# B&R Automation Studio project SimuladorTesis
Automation Studio 4.8.2.72; technology packages: mapp 5.8.0

## Configuration Config1

CPU X20CP1584, AutomationRuntime C4.90, Build 4.1.2, Safety 0.0, Vc V4.72.2

### Task classes (Cpu.sw)
```
Cyclic#2:
  MainLogic <- Source.MachineSimulation.MainLogic.prg
  OEECalc <- Source.MachineSimulation.OEECalc.prg
Cyclic#3:
  VisCtrl <- Source.Visualization.VisCtrl.prg
VcDataObjects: Visu <- Source.Visualization.Visu.dob
Binaries: vcctext, arialbd, vccpiech, vcmgr, vccpopup, vcxml, vccdt, vccshape, vcchspot, vcnet, vcdsloc, vcbclass, vcfntttf, Visu01, arsvcreg, vctcal, Visu03, vcshared, vcrt, vcpkat, vccbmp, TCData, vcfile, vccbtn, vccnum, vccddbox, vccslider, vcalarm, vcpdsw, FWRules, vcdsint, arial, vccovl, udbdef, vccscale, vccline, vcpdvnc, vcpfar00, vccalarm, vccstr, vcchtml, vcctrend, vcgclass, vcclbox, vccurl, Visu02, OEE, PackML, Role, arconfig, User, asfw, ashwd, ashwac, sysconf, iomap, Config
Libraries: MpPackML, MpBase, astime, runtime, LoopCont, sys_lib, brsystem, standard, MpWebXs, AsArSdm, MpOee, asieccon, fileio, dataobj, vcresman
```

### Hardware
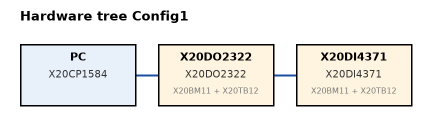
```
PC : X20CP1584 v1.8.1.0
  Connector IF1:
    ActivateIna = 0
  Connector IF2:
    ActivateDevice = 1
    Mode = Manual
    InternetAddress = 192.168.0.20
    SubnetMask = 255.255.255.0
    InaPort = 11160
    Vnc1
    VncVcObjectName1 = Visu
    VncKeyMappingFile1 = VC\PS2-Keyboard.dis
    VncRefreshRate1 = 250
  ConfigurationID = SimuladorTesis_Config1
  FileDevice1
  FileDeviceName1 = Historico
  FileDevicePath1 = C:\Historico
X20BM11 : X20BM11 v1.0.0.1  [X2X1 -> PC.IF6]
X20BM11a : X20BM11 v1.0.0.1  [X2X1 -> X20BM11.X2X2]
X20DI4371 : X20DI4371 v1.1.0.0  [SS1 -> X20TB12a.SS; SL -> X20BM11a.SL1]
X20DO2322 : X20DO2322 v1.1.0.0  [SS1 -> X20TB12.SS; SL -> X20BM11.SL1]
X20TB12 : X20TB12 v1.0.0.0
X20TB12a : X20TB12 v1.0.0.0
```

### IoMap.iom - PC/IoMap.iom
```iecst
VAR_CONFIG
	::paro AT %IX."X20DI4371".DigitalInput01;
END_VAR
```

### OEE.mpoeecore - PC/mappServices/OEE.mpoeecore
```
Element gOeeCore (Type=mpoeecore)
  Oee:
    Shifts:
      [0]:
        Name = Morning
        TotalTime:
          Start = 21600000
          End = 50400000
        ScheduledDowntime:
          [0]:
            Reason = Lunch
            Start = 39600000
            End = 41400000
      [1]:
        Name = Afternoon
        TotalTime:
          Start = 50400000
          End = 79200000
        ScheduledDowntime:
          [0]:
            Reason = Dinner
            Start = 64800000
            End = 66600000
  Alarms = MpAlarmX
```

### PackML.mppackmlcore - PC/mappServices/PackML.mppackmlcore
```
Element gPackMLCore (Type=mppackmlcore)
  Modes:
    Mode[1]:
      ModeID = 1
      Name = Production
      State[5] = 0
      State[10] = 0
      State[11] = 0
      State[12] = 0
      State[13] = 0
      State[14] = 0
      State[16] = 0
      State[17] = 0
    Mode[2]:
      ModeID = 2
      Name = Mode[3]
      State[5] = 0
      State[10] = 0
      State[11] = 0
      State[12] = 0
      State[13] = 0
      State[14] = 0
  Alarms = MpAlarmX
```

## Logical view

Binary libraries used (declarations not repeated): operator, runtime, astime, AsIecCon, LoopCont, sys_lib, brsystem, standard, AsArSdm, MpOee 5.14.1, MpBase 5.08.0, MpWebXs 5.08.0, MpPackML 5.14.1

### Global.var - Global variables
```iecst
VAR
	paro : BOOL;
	piezasProducidasTotales : DINT;
	piezasProducidas : DINT;
	piezasRechazadas : DINT;
	tiempoDeCiclo : REAL;
END_VAR
```


### Program Logical/Source/MachineSimulation/MainLogic (IEC)

#### Main.st - Init, cyclic, exit code
```iecst
PROGRAM _INIT
	(* Insert code here *)
	mpPackMLCore_Simulador.Enable := TRUE;
	mpPackMLCore_Simulador.MpLink := ADR(gPackMLCore);
	mpPackMLMode_Simulador.Enable := TRUE;
	mpPackMLMode_Simulador.MpLink := ADR(gPackMLCore);
	mpPackMLMode_Simulador.ModeID := 1;

	RTInfo_0(enable := TRUE);

	tiempoCiclo := 5;

	//Se pasa la variable local a la global
	tiempoDeCiclo := tiempoCiclo;

	//Escondiendo los pop up's
	idlePopUpStatus 			 := HIDE;
	maintenancePopUpStatus	     := HIDE;
	maintenanceTimeBalloonStatus := HIDE;

END_PROGRAM

PROGRAM _CYCLIC

	//Se pasa la variable local a la global
	tiempoDeCiclo := tiempoCiclo;

	DTStructureGetTime_0(enable := TRUE, pDTStructure := ADR(sysTime));

	CASE mpPackMLCore_Simulador.StateCurrent OF

		mpPACKML_STATE_UNDEFINED:

			mpPackMLMode_Simulador.Activate := TRUE;

		mpPACKML_STATE_IDLE:

			//Llamando a la acción para aparecer al pop up de paro
			IdlePopUpWindow;

		mpPACKML_STATE_STARTING:

			//Limpiando los datos del pop up de paro
			CleanPopUpData;

			mpPackMLMode_Simulador.Start 		 := FALSE;
			mpPackMLMode_Simulador.StateComplete := TRUE;

		mpPACKML_STATE_EXECUTE:

			(* Acumuladores de tiempo *)
			tiempoEnProduccion := tiempoEnProduccion + (UDINT_TO_REAL(RTInfo_0.cycle_time)/1000000);
			cuentaTiempo 	   := cuentaTiempo + (UDINT_TO_REAL(RTInfo_0.cycle_time)/1000000);

			IF cuentaTiempo >= tiempoCiclo THEN

				cuentaTiempo := 0;

				IF NOT TON_rechazada.IN THEN
					random 				           := ((sysTime.millisec*sysTime.second*(sysTime.minute+5)/(sysTime.hour+3)+17)*3); //Generando un numero pseudo aleatorio
					rejected 			           := REAL_TO_SINT(random);
					banderaRandomRechazada         := ABS(rejected);
					banderaRandomRechazada_Milisec := SINT_TO_UINT(banderaRandomRechazada)*MS_FACTOR;
					TON_rechazada.PT               := UINT_TO_TIME(banderaRandomRechazada_Milisec);
					TON_rechazada.IN               := TRUE; //Activando el timer para lanzar una pieza rechazada
				END_IF

				IF TON_rechazada.Q THEN
					TON_rechazada.IN := FALSE;
					TON_rechazada(); //Llamando al timer de rechazo
					piezasRechazadas := piezasRechazadas + 1;
				ELSE
					piezasProducidas := piezasProducidas + 1;
				END_IF;
			END_IF;

			TON_rechazada(); //Llamando al timer de rechazo

		mpPACKML_STATE_STOPPING:

			TON_rechazada.IN    				 := FALSE;
			TON_rechazada();
			cuentaTiempo 						 := 0;
			mpPackMLMode_Simulador.Stop			 := FALSE;
			mpPackMLMode_Simulador.StateComplete := TRUE;

		mpPACKML_STATE_STOPPED:

			//Llamando a la acción para aparecer al pop up de paro
			IdlePopUpWindow;

		mpPACKML_STATE_RESETTING:

			//Limpiando los datos del pop up de paro
			CleanPopUpData;

			mpPackMLMode_Simulador.Reset		 := FALSE;
			mpPackMLMode_Simulador.StateComplete := TRUE;

		mpPACKML_STATE_ABORTING:

			TON_rechazada.IN    				 := FALSE;
			TON_rechazada();
			cuentaTiempo 						 := 0;
			mpPackMLMode_Simulador.Abort		 := FALSE;
			mpPackMLMode_Simulador.StateComplete := TRUE;

		mpPACKML_STATE_CLEARING:

			mpPackMLMode_Simulador.Clear		 := FALSE;
			mpPackMLMode_Simulador.StateComplete := TRUE;

	END_CASE;

	//Contador general de piezas producidas
	piezasProducidasTotales := piezasProducidas + piezasRechazadas;

	mpPackMLMode_Simulador();
	mpPackMLCore_Simulador();

	//Actualizando el comando de estado completo con un flanco positivo
	IF mpPackMLMode_Simulador.StateComplete AND (mpPackMLMode_Simulador.StateComplete <> OldStateComplete) THEN
		mpPackMLMode_Simulador.StateComplete := FALSE;
	END_IF;
	OldStateComplete := mpPackMLMode_Simulador.StateComplete;

	(* VISU CONTROL *)
	IF openMaintenanceTimeDetails THEN

		maintenanceTimeBalloonStatus := SHOW;

	ELSE

		maintenanceTimeBalloonStatus := HIDE;

	END_IF;

END_PROGRAM

PROGRAM _EXIT

	mpPackMLCore_Simulador.Enable := FALSE;
	mpPackMLCore_Simulador();
	mpPackMLMode_Simulador.Enable := FALSE;
	mpPackMLMode_Simulador();

END_PROGRAM
```

#### Variables.var - Local variables
```iecst
VAR
	mpPackMLCore_Simulador : MpPackMLCore;
	mpPackMLMode_Simulador : MpPackMLMode;
	OldStateComplete : BOOL;
	DTStructureGetTime_0 : DTStructureGetTime;
	sysTime : DTStructure;
	random : REAL;
END_VAR
VAR RETAIN
	tiempoCiclo : REAL;
END_VAR
VAR
	RTInfo_0 : RTInfo;
	cuentaTiempo : REAL;
	rejected : SINT;
	idlePopUpStatus : USINT;
	maintenanceTimeBalloonStatus : USINT;
	maintenancePopUpStatus : USINT;
END_VAR
(*BANDERAS DEL SISTEMA*)
VAR
	banderaRandomRechazada : SINT;
	banderaRandomRechazada_Milisec : UINT;
	aceptarTiempoRetrabajo : BOOL;
	aceptarTiempoMantto : BOOL;
	aceptarManttoPredict : BOOL;
	aceptarManttoAutonomo : BOOL;
	openMaintenanceTimeDetails : BOOL;
END_VAR
(*TEMPORIZADORES DEL SISTEMA*)
VAR
	TON_rechazada : TON;
	TON_Idle_PopUp : {REDUND_UNREPLICABLE} TON;
	TON_Idle_TimeDelay : TON;
	TON_Mantto_TimeDelay : TON;
END_VAR
(*ACUMULADORES DE TIEMPO *)
VAR
	tiempoOcioso : REAL;
	tiempoRetrabajo : REAL;
	tiempoManttoTotal : REAL;
	tiempoManttoPredict : REAL;
	tiempoManttoAutonomo : REAL;
	tiempoEnProduccion : REAL;
END_VAR
(*CONSTANTES DEL SISTEMA*)
VAR CONSTANT
	SHOW : USINT := 0;
	HIDE : USINT := 1;
	MS_FACTOR : UINT := 1000;
	POP_UP_TIMER : TIME := T#20S;
	IDLE_DELAY_TIME : TIME := T#20S;
END_VAR
VAR
	manttoPredictSelected : BOOL;
	manttoAutonomoSelected : BOOL;
END_VAR
```

#### IdlePopUp.st
```iecst
ACTION IdlePopUpWindow:

	TON_Idle_PopUp(IN := TRUE , PT := POP_UP_TIMER);

	IF TON_Idle_PopUp.Q THEN
		//Se muestra el pop up de paro
		idlePopUpStatus := SHOW;
		TON_Idle_TimeDelay(IN := TRUE , PT := IDLE_DELAY_TIME); //Comienza el retardo de cierre del pop-up
		(*El usuario decide en que acumulador se contará el tiempo de paro*)
		//PARO POR RETRABAJO
		IF aceptarTiempoRetrabajo THEN

			TON_Idle_TimeDelay(IN := FALSE);
			tiempoRetrabajo := tiempoRetrabajo + (UDINT_TO_REAL(RTInfo_0.cycle_time)/1000000);
			idlePopUpStatus := HIDE;
			//PARO POR MANTENIMIENTO PROGRAMADO
		ELSIF aceptarTiempoMantto THEN

			TON_Idle_TimeDelay(IN := FALSE);
			TON_Mantto_TimeDelay(IN := TRUE , PT := IDLE_DELAY_TIME); //Comienza el retardo de cierre del pop-up

			idlePopUpStatus        := HIDE;
			maintenancePopUpStatus := SHOW;

			IF manttoPredictSelected THEN

				TON_Mantto_TimeDelay(IN := FALSE);
				tiempoManttoPredict    := tiempoManttoPredict + (UDINT_TO_REAL(RTInfo_0.cycle_time)/1000000);
				maintenancePopUpStatus := HIDE;

			ELSIF manttoAutonomoSelected THEN

				TON_Mantto_TimeDelay(IN := FALSE);
				tiempoManttoAutonomo   := tiempoManttoAutonomo + (UDINT_TO_REAL(RTInfo_0.cycle_time)/1000000);
				maintenancePopUpStatus := HIDE;

			ELSIF TON_Mantto_TimeDelay.Q THEN
				tiempoOcioso 	:= tiempoOcioso + (UDINT_TO_REAL(RTInfo_0.cycle_time)/1000000);
			END_IF;

			tiempoManttoTotal 	:= tiempoManttoAutonomo + tiempoManttoPredict;

			//PARO DE TIEMPO OCIOSO
		ELSIF TON_Idle_TimeDelay.Q THEN
			tiempoOcioso 	:= tiempoOcioso + (UDINT_TO_REAL(RTInfo_0.cycle_time)/1000000);
		END_IF;
	END_IF;

END_ACTION
```

#### CleanPopUpData.st
```iecst
ACTION CleanPopUpData:

	//Reset del temporizador para el pop up
	TON_Idle_PopUp(IN := FALSE);
	TON_Mantto_TimeDelay(IN := FALSE);
	TON_Idle_TimeDelay(IN  := FALSE);
	aceptarTiempoRetrabajo := FALSE;
	aceptarTiempoMantto	   := FALSE;
	manttoAutonomoSelected := FALSE;
	manttoPredictSelected  := FALSE;

END_ACTION
```

### Program Logical/Source/MachineSimulation/MainLogicFBD (IEC)

#### Cyclic.fbd - Cyclic code
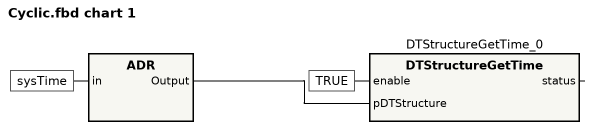
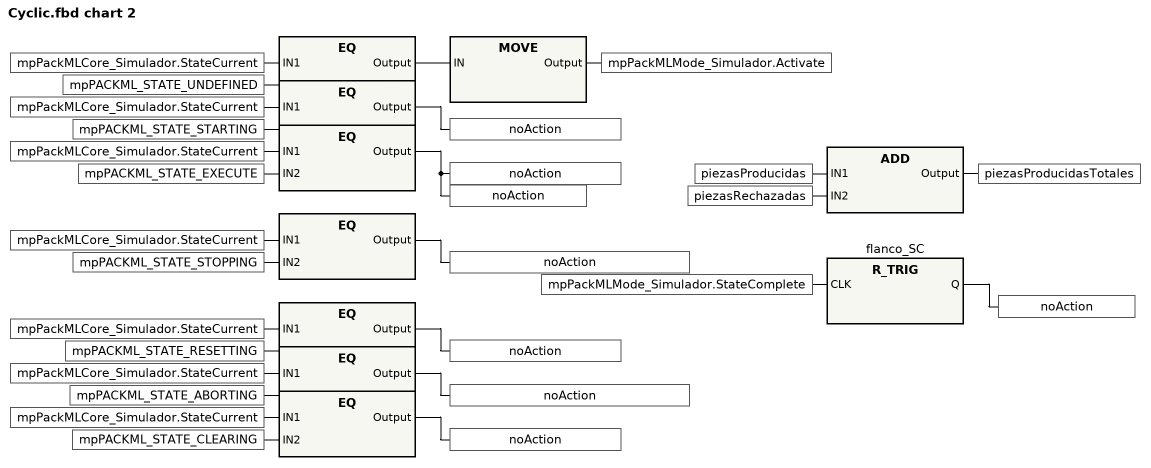
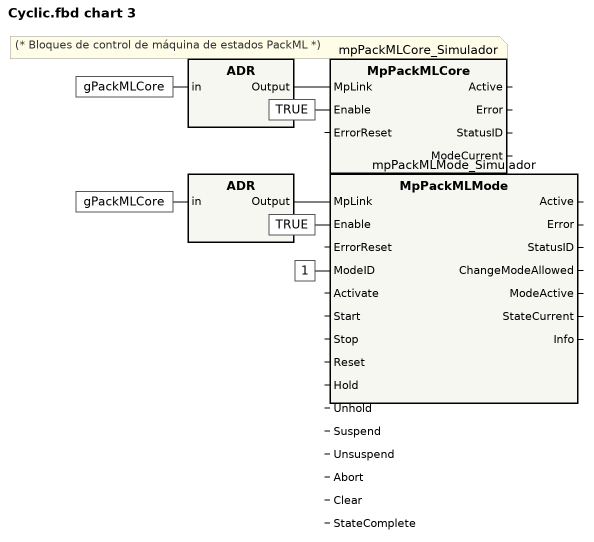
Diagram, in the editor's own instruction-list form stored in the file:
```il
PROGRAM _CYCLIC
(* Bloques de control de máquina de estados PackML *)
VAR
	zz0000FCT_1_1_ADR_Output : UDINT;
	zz0000FCT_2_1_EQ_Output : BOOL;
	zz0000FCT_2_8_EQ_Output : BOOL;
	zz0000FCT_2_3_EQ_Output : BOOL;
	zz0000FCT_2_4_EQ_Output : BOOL;
	zz0000FCT_2_5_EQ_Output : BOOL;
	zz0000FCT_2_7_EQ_Output : BOOL;
	zz0000FCT_2_6_EQ_Output : BOOL;
	FinalizarTransicion_$$$$$$ : SFCActionType;
	CuentaTiempo_$$$$$$ : SFCActionType;
	CicloProceso_$$$$$$ : SFCActionType;
	ConfirmarProcesoDetenido_$$$$$$ : SFCActionType;
	ResetSC_$$$$$$ : SFCActionType;
	zz0000FCT_3_2_ADR_Output : UDINT;
	zz0000FCT_3_1_ADR_Output : UDINT;
END_VAR

{NetworkNumber := 1}
LD sysTime
ADR
ST zz0000FCT_1_1_ADR_Output
LD TRUE
ST DTStructureGetTime_0.enable
LD zz0000FCT_1_1_ADR_Output
ST DTStructureGetTime_0.pDTStructure
CAL DTStructureGetTime_0

{NetworkNumber := 2}
LD mpPackMLCore_Simulador.StateCurrent
EQ mpPACKML_STATE_UNDEFINED
ST zz0000FCT_2_1_EQ_Output
LD mpPackMLCore_Simulador.StateCurrent
EQ mpPACKML_STATE_STARTING
ST zz0000FCT_2_8_EQ_Output
LD zz0000FCT_2_8_EQ_Output
S FinalizarTransicion_$$$$$$.AC.P
LD mpPackMLCore_Simulador.StateCurrent
EQ mpPACKML_STATE_EXECUTE
ST zz0000FCT_2_3_EQ_Output
LD zz0000FCT_2_3_EQ_Output
S CuentaTiempo_$$$$$$.AC.N
LD zz0000FCT_2_3_EQ_Output
S CicloProceso_$$$$$$.AC.N
LD mpPackMLCore_Simulador.StateCurrent
EQ mpPACKML_STATE_STOPPING
ST zz0000FCT_2_4_EQ_Output
LD zz0000FCT_2_4_EQ_Output
S ConfirmarProcesoDetenido_$$$$$$.AC.P
LD mpPackMLCore_Simulador.StateCurrent
EQ mpPACKML_STATE_RESETTING
ST zz0000FCT_2_5_EQ_Output
LD zz0000FCT_2_5_EQ_Output
S FinalizarTransicion_$$$$$$.AC.P
LD mpPackMLCore_Simulador.StateCurrent
EQ mpPACKML_STATE_ABORTING
ST zz0000FCT_2_7_EQ_Output
LD zz0000FCT_2_7_EQ_Output
S ConfirmarProcesoDetenido_$$$$$$.AC.P
LD mpPackMLCore_Simulador.StateCurrent
EQ mpPACKML_STATE_CLEARING
ST zz0000FCT_2_6_EQ_Output
LD zz0000FCT_2_6_EQ_Output
S FinalizarTransicion_$$$$$$.AC.P
LD zz0000FCT_2_1_EQ_Output
MOVE
ST mpPackMLMode_Simulador.Activate
LD piezasProducidas
ADD piezasRechazadas
ST piezasProducidasTotales
LD mpPackMLMode_Simulador.StateComplete
ST flanco_SC.CLK
CAL flanco_SC
LD flanco_SC.Q
S ResetSC_$$$$$$.AC.N

{NetworkNumber := 3}
LD gPackMLCore
ADR
ST zz0000FCT_3_2_ADR_Output
LD gPackMLCore
ADR
ST zz0000FCT_3_1_ADR_Output
LD zz0000FCT_3_2_ADR_Output
ST mpPackMLCore_Simulador.MpLink
LD TRUE
ST mpPackMLCore_Simulador.Enable
CAL mpPackMLCore_Simulador
LD zz0000FCT_3_1_ADR_Output
ST mpPackMLMode_Simulador.MpLink
LD TRUE
ST mpPackMLMode_Simulador.Enable
LD 1
ST mpPackMLMode_Simulador.ModeID
CAL mpPackMLMode_Simulador

END_PROGRAM
```

#### Init.fbd - Initialization code
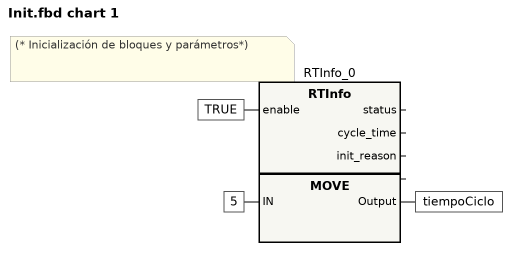
Diagram, in the editor's own instruction-list form stored in the file:
```il
PROGRAM _INIT
(* Inicialización de bloques y parámetros *)

{NetworkNumber := 1}
LD TRUE
ST RTInfo_0.enable
CAL RTInfo_0
LD 5
MOVE
ST tiempoCiclo

END_PROGRAM
```

#### Variables.var - Local variables
```iecst
VAR
	mpPackMLCore_Simulador : MpPackMLCore;
	mpPackMLMode_Simulador : MpPackMLMode;
	DTStructureGetTime_0 : DTStructureGetTime;
	sysTime : DTStructure;
	random : REAL;
	tiempoCiclo : REAL;
	RTInfo_0 : RTInfo;
	cuentaTiempo : REAL;
	TON_rechazada : TON;
	banderaRandomRechazada_Milisec : UINT;
END_VAR
VAR CONSTANT
	MS_FACTOR : UINT := 1000;
END_VAR
VAR
	tiempoCicloREAL : REAL;
	tiempoCicloTerminado : BOOL;
	banderaRandomRechazadaUINT : UINT;
	iniciarTimer : BOOL;
	valorTimer : TIME;
	timerFinalizado : BOOL;
	flanco_SC : R_TRIG;
	contarRechazo : BOOL;
	resetRechazo : BOOL;
END_VAR
```

#### CuentaTiempo.ld
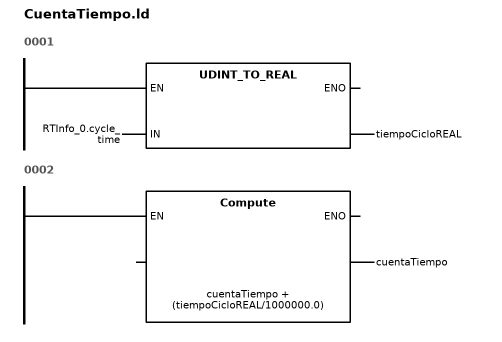
Ladder, written as Structured Text:
```iecst
ACTION CuentaTiempo:
(* Network 1 *)
tiempoCicloREAL := UDINT_TO_REAL(RTInfo_0.cycle_time);

(* Network 2 *)
cuentaTiempo := cuentaTiempo + (tiempoCicloREAL/1000000.0);
END_ACTION
```

#### CicloProceso.ld
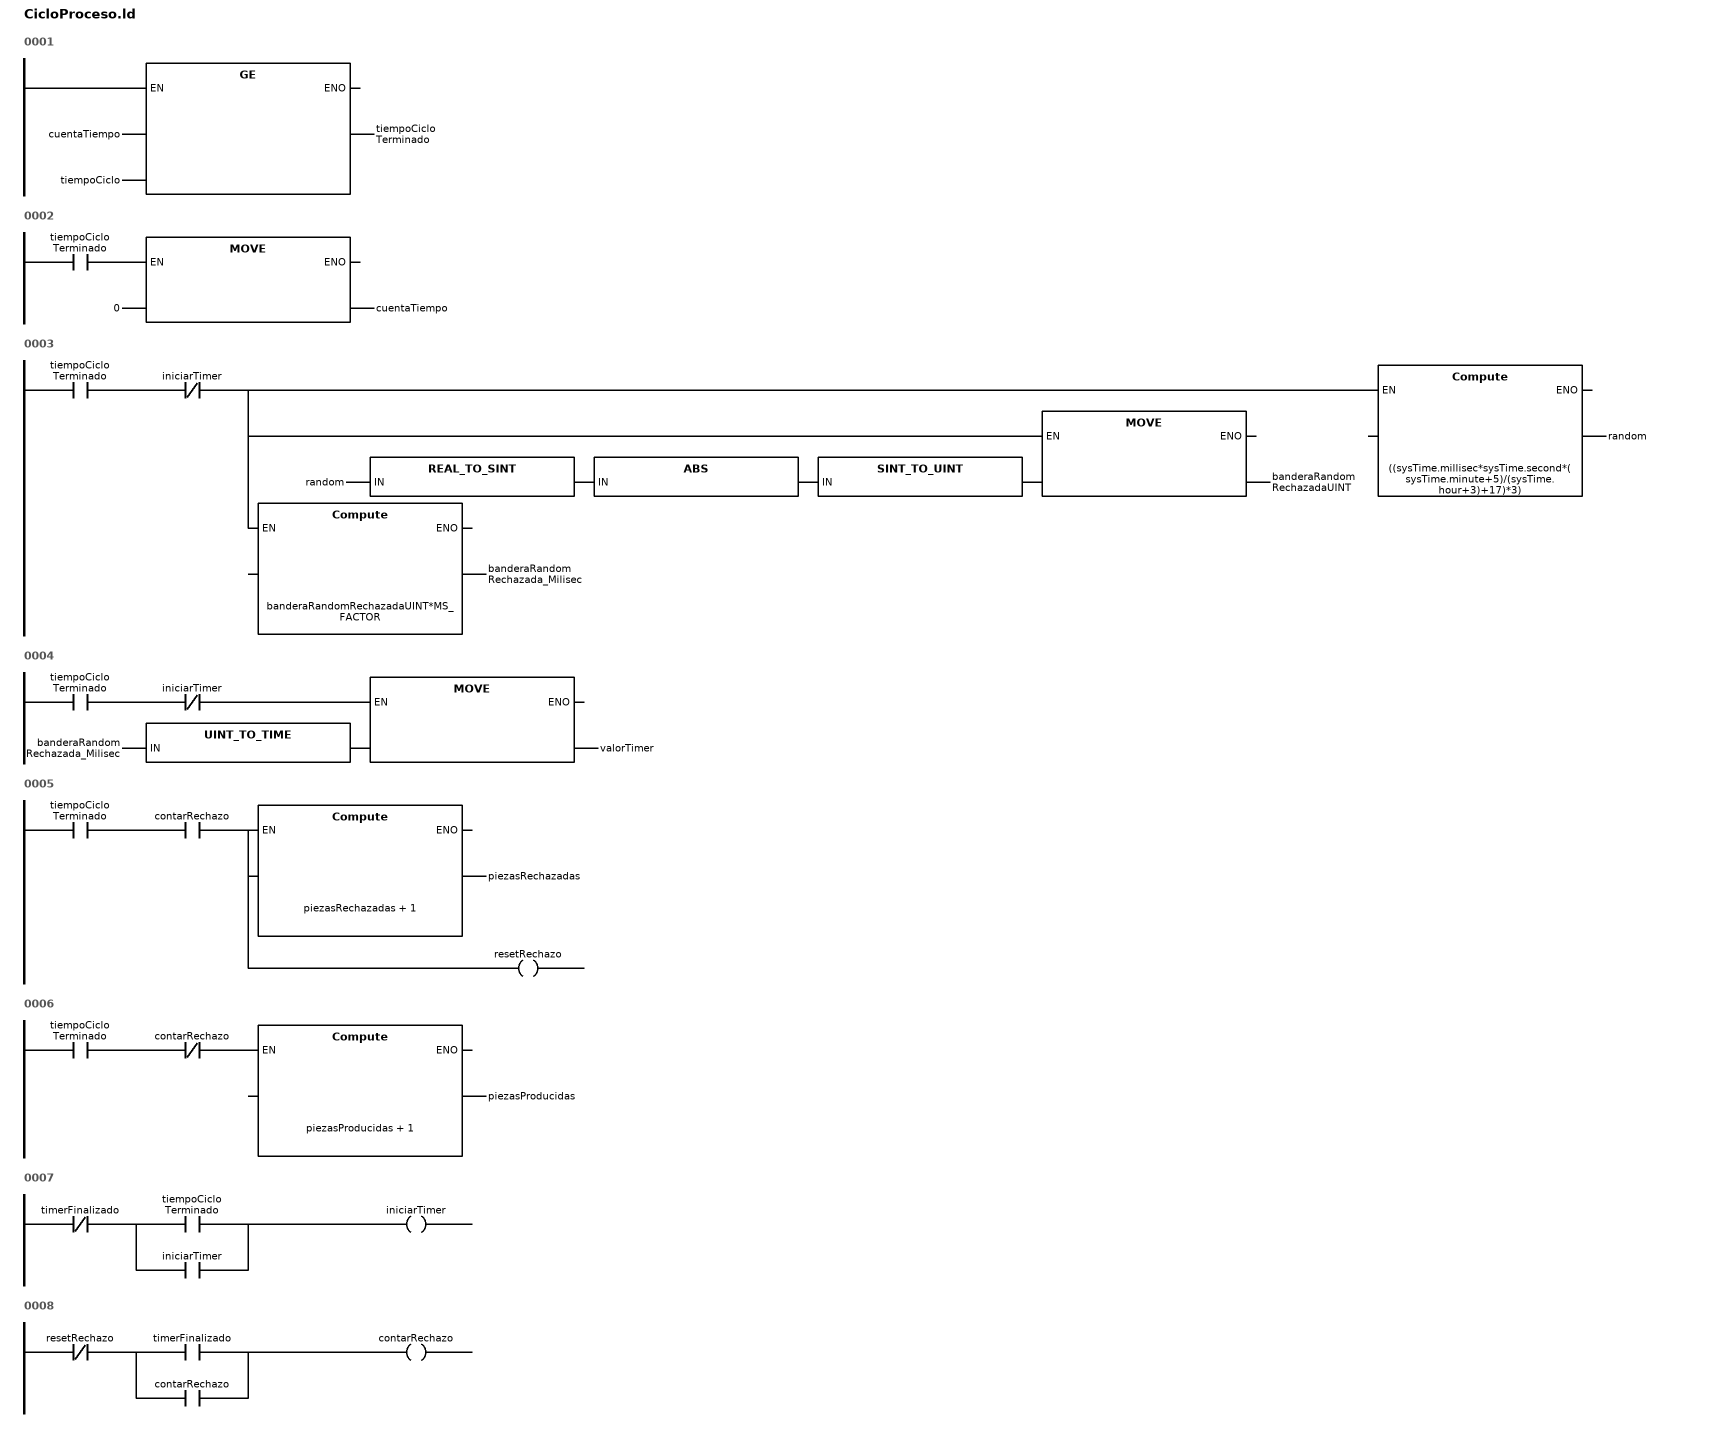
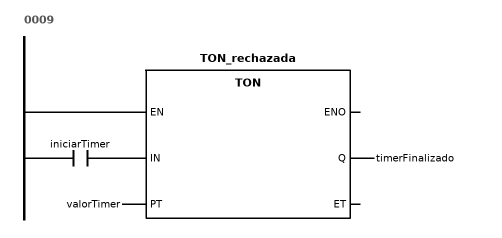
Ladder, written as Structured Text:
```iecst
ACTION CicloProceso:
(* Network 1 *)
tiempoCicloTerminado := cuentaTiempo >= tiempoCiclo;

(* Network 2 *)
IF tiempoCicloTerminado THEN cuentaTiempo := 0; END_IF;

(* Network 3 *)
IF tiempoCicloTerminado AND NOT iniciarTimer THEN
    random := ((sysTime.millisec*sysTime.second*(sysTime.minute+5)/(sysTime.hour+3)+17)*3);
    banderaRandomRechazadaUINT := SINT_TO_UINT(ABS(REAL_TO_SINT(random)));
    banderaRandomRechazada_Milisec := banderaRandomRechazadaUINT*MS_FACTOR;
END_IF;

(* Network 4 *)
IF tiempoCicloTerminado AND NOT iniciarTimer THEN
    valorTimer := UINT_TO_TIME(banderaRandomRechazada_Milisec);
END_IF;

(* Network 5 *)
IF tiempoCicloTerminado AND contarRechazo THEN piezasRechazadas := piezasRechazadas + 1; END_IF;
resetRechazo := tiempoCicloTerminado AND contarRechazo;

(* Network 6 *)
IF tiempoCicloTerminado AND NOT contarRechazo THEN piezasProducidas := piezasProducidas + 1; END_IF;

(* Network 7 *)
iniciarTimer := NOT timerFinalizado AND (tiempoCicloTerminado OR iniciarTimer);

(* Network 8 *)
contarRechazo := NOT resetRechazo AND (timerFinalizado OR contarRechazo);

(* Network 9 *)
TON_rechazada(IN := iniciarTimer, PT := valorTimer);
timerFinalizado := TON_rechazada.Q;
END_ACTION
```

#### ConfirmarProcesoDetenido.ld
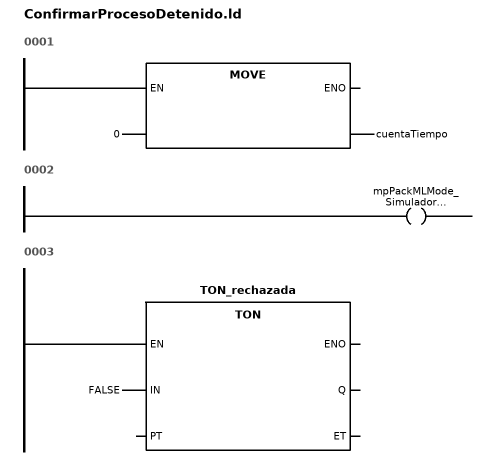
Ladder, written as Structured Text:
```iecst
ACTION ConfirmarProcesoDetenido:
(* Network 1 *)
cuentaTiempo := 0;

(* Network 2 *)
mpPackMLMode_Simulador.StateComplete := TRUE;

(* Network 3 *)
TON_rechazada(IN := FALSE);
END_ACTION
```

#### FinalizarTransicion.ld
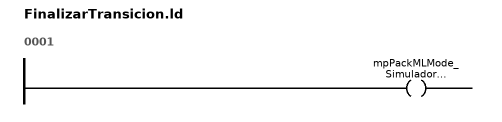
Ladder, written as Structured Text:
```iecst
ACTION FinalizarTransicion:
(* Network 1 *)
mpPackMLMode_Simulador.StateComplete := TRUE;
END_ACTION
```

#### ResetSC.ld
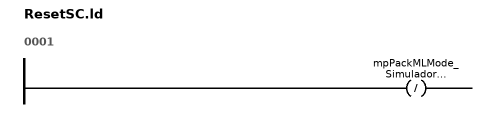
Ladder, written as Structured Text:
```iecst
ACTION ResetSC:
(* Network 1 *)
mpPackMLMode_Simulador.StateComplete := FALSE;
END_ACTION
```

### Program Logical/Source/MachineSimulation/Program3 (IEC)

#### Cyclic.ld - Cyclic code
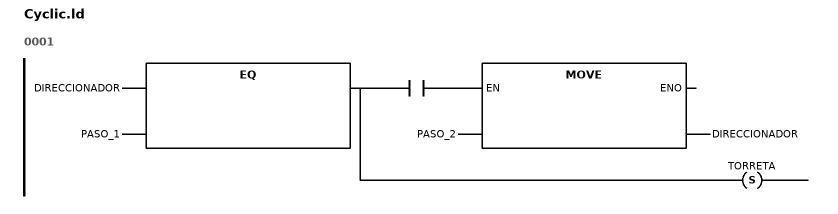
Ladder, written as Structured Text:
```iecst
PROGRAM _CYCLIC
VAR
    _t1 : BOOL;
END_VAR
(* Network 1 *)
_t1 := DIRECCIONADOR = PASO_1;
IF _t1 AND () THEN DIRECCIONADOR := PASO_2; END_IF;
IF _t1 THEN TORRETA := TRUE; END_IF;
END_PROGRAM
```

#### Variables.var - Local variables
```iecst
VAR CONSTANT
	PASO_1 : INT := 10;
END_VAR
VAR
	DIRECCIONADOR : INT;
	TORRETA : BOOL;
END_VAR
VAR CONSTANT
	PASO_2 : INT := 20;
END_VAR
```

### Program Logical/Source/MachineSimulation/OEECalc (IEC)

#### Variables.var
```iecst
VAR
	MpOeeCore_Simulador : MpOeeCore;
	OeeParam : MpOeeCoreParType;
END_VAR
```

#### Main.st
```iecst
PROGRAM _INIT

	MpOeeCore_Simulador.Enable     := TRUE;
	MpOeeCore_Simulador.DeviceName := ADR('Historico');
	MpOeeCore_Simulador.MpLink     := ADR(gOeeCore);
	OeeParam.IdealCycleTime		   := REAL_TO_TIME(tiempoDeCiclo)*1000;
	MpOeeCore_Simulador.Parameters := ADR(OeeParam);

END_PROGRAM

PROGRAM _CYCLIC

	//Registrando un paro de máquina
	IF (MpPackMLStateCurrent(gPackMLCore) <> mpPACKML_STATE_EXECUTE) THEN
		MpOeeCore_Simulador.Downtime := TRUE;
	ELSE
		MpOeeCore_Simulador.Downtime := FALSE;
	END_IF;

	MpOeeCore_Simulador.PieceCounter  := piezasProducidasTotales;
	MpOeeCore_Simulador.RejectCounter := piezasRechazadas;
	MpOeeCore_Simulador();

END_PROGRAM

PROGRAM _EXIT

	MpOeeCore_Simulador(Enable := FALSE);

END_PROGRAM
```

- Visualisation Logical/Source/Visualization (not shown)

Listed in the project but not available here: Logical/Global.typ, Logical/Source/MachineSimulation/MainLogic/Types.typ, Logical/Source/MachineSimulation/MainLogicFBD/Exit.fbd, Logical/Source/MachineSimulation/MainLogicFBD/Types.typ, Logical/Source/MachineSimulation/Program3/Init.ld, Logical/Source/MachineSimulation/Program3/Exit.ld, Logical/Source/MachineSimulation/Program3/Types.typ
